// TIA Portal V16 export
// export: Created 2025-10-07T21:39:08.1582299Z, ExportSetting WithDefaults, DisplayName Totally Integrated Automation Portal, DisplayVersion V16, DisplayName TIA Portal Version Control Interface, DisplayVersion V16, DisplayName TIA Portal Openness, DisplayVersion V16, DisplayName STEP 7 Professional, DisplayVersion V16, DisplayName STEP 7 Safety, DisplayVersion V16, DisplayName WinCC Advanced, DisplayVersion V16
DATA_BLOCK "PositionManagement"   // DB51
VERSION : 0.1
// stored: AutoNumber true, IsOnlyStoredInLoadMemory false, IsWriteProtectedInAS false
   VAR RETAIN
      Data : Struct   // Data
         CntPlsPrev : DInt := 0;   // Flowpulsen vorige scan
         CntPlsDiff : DInt := 0;   // Flowpulsen verschil
         CntPlsAct : DInt := 0;   // Flowpulsen actueel
         DosActueel : Real := 0.0;   // Dosering actueel (not used)
         Actual_Axis3_Position : Real;   // Actual Position of Axis 3 stored in this datablock
         Actual_Axis1_Position : Real;
      END_STRUCT;
      "Axis 3" : Struct
         Values : Struct
            AxisName : String := 'Drive 3 - Wals';
            "Reference Position" : Int := 0;
            "Set Position" : Real := -50.0;
            "Rest Position" : Real := -25.0;
            Acceleration : Real := 0.0;
            Deacceleration : Real;
            "Axis Correction" : Real := 1.0E-06;
            "Position Offset" : Real := 35.0;
            Pulsfactor : Real := 0.82;
            Axis_Speed : Int := 0;
            ModuloFactor : Real := 360.0;
         END_STRUCT;
         Commands : Struct
            "Go To Rest" : Bool;
            "Start Ref Run" : Bool;
            "Take Over Pos" : Bool;
            "Go To Position" : Bool;
            "Jog Fwd" : Bool;
            "Jog Rev" : Bool;
            Axis_Brake : Bool;
            MasterWord : String;
            "Master Callback" : String;
         END_STRUCT;
         Messages : Struct
            "Axis Busy" : Bool;
            "Error Executing Command" : Bool;
            "Axis On Rest" : Bool;
            "Axis On Position" : Bool;
            "Drive State (Option)" : String;
            "Slip State" : String;
            AxisHasReference : Bool;
         END_STRUCT;
      END_STRUCT;
      Demo_Pos : Struct
         Desired_Pos : Real;
         Start : Bool;
         SetRefRunActive : Bool;
         RequestMove1 : Bool;
         RequestMove2 : Bool;
         PositionMove2 : Real := -50.0;
         PositionMove1 : Real := -250.0;
         Pos2Done : Bool;
         BrakeOnPos1 : Bool;
         BrakeOnPos2 : Bool;
         ManualSensorOverride : Bool;
      END_STRUCT;
      Axis_1 : Struct
         Values : Struct
            AxisName : String := 'Drive 1 - Infeed';
            "Reference Position" : Int := 0;
            "Set Position" : Real := 0.0;
            "Rest Position" : Real := 0.0;
            Acceleration : Real := 0.0;
            Deacceleration : Real;
            "Axis Correction" : Real := 1.0E-06;
            "Position Offset" : Real := 0.001;
            Pulsfactor : Real := -0.359;
            Axis_Speed : Int := 0;
            LimitEncValue : DInt := 0;
         END_STRUCT;
         Commands : Struct
            "Go To Rest" : Bool;
            "Start Ref Run" : Bool;
            "Take Over Pos" : Bool;
            "Go To Position" : Bool;
            "Jog Fwd" : Bool;
            "Jog Rev" : Bool;
            Axis_Brake : Bool;
            ReferenceSwitch : Bool;
            MasterWord : String;
            "Master Callback" : String;
         END_STRUCT;
         Messages : Struct
            "Axis Busy" : Bool;
            "Error Executing Command" : Bool;
            "Axis On Rest" : Bool;
            "Axis On Position" : Bool;
            "Drive State (Option)" : String;
            "Slip State" : String;
            AxisHasReferenceDelayed : Bool;
            AxisHasReference : Bool;
            SetAxisHasRefFromEnc : Bool;
            MaxOverflowValueDint : DInt := 16#8261A800;
         END_STRUCT;
      END_STRUCT;
   END_VAR
BEGIN
END_DATA_BLOCK
